PROGRAM Simulation
VAR
	_CylinderDistance		:REAL;
END_VAR

GVL._Cylinder.CylinderDistance := _CylinderDistance;

IF GVL._Cylinder.Extend THEN
	_CylinderDistance := _CylinderDistance + 0.1;
ELSIF GVL._Cylinder.Retract THEN
	_CylinderDistance := _CylinderDistance - 0.1;
END_IF

END_PROGRAM

(* stored: Version 1.1.0.1
   POU Simulation: Id {f642e345-0ca8-4a57-a78d-e726bf0c6a88}, SpecialFunc None *)
